Fanuc KAREL source: kt00946.KL

-- PROVISIONAL review KL for V1013-1; original PC SHA256 d5fd0a12249a2da244c6201568b32e45ecb654f153b10b2fbbc033967bf3bbc0
-- Incomplete behavior may be omitted. Consult companion uncertainty JSON. Do not deploy.
PROGRAM KT00946
%NOLOCKGROUP
VAR
  ENTRY : INTEGER
  PNAME : STRING[80]
  VNAME : STRING[80]
  STATUS : INTEGER
-- UNRESOLVED_DECL VALUE type=002011
BEGIN
  -- UNRESOLVED_PC offsets 5-12; opcodes 9C,23
  -- UNRESOLVED_PC offsets 17-25; opcodes 3F,75
  -- UNRESOLVED_PC offsets 30-43; opcodes 3F,75
  -- UNRESOLVED_PC offsets 48-86; opcodes 27,22,22,2A,22,2A,22,22,AF
  -- UNRESOLVED_PC offsets 91-95; opcodes 7F
END KT00946
